FUNCTION TryConvert_STRING_TO_TOD : BOOL
VAR_INPUT
	in : STRING;
	out : REFERENCE TO TOD;
END_VAR

IF in <> TOD_TO_STRING(STRING_TO_TOD(in)) THEN
	RETURN;
END_IF

out := STRING_TO_TOD(in);
TryConvert_STRING_TO_TOD := TRUE;

END_FUNCTION

(* stored: Version 1.1.0.1, ProductVersion 3.1.4024.12
   POU TryConvert_STRING_TO_TOD: Id {3554b624-6e3b-4daa-93d6-53c19dcde729}, SpecialFunc None *)
